TYPE ST_pcmChillerDefaultParameters :
STRUCT
	aSetPointLimitsTemperature : ARRAY[1..2] OF REAL := [10,28];
END_STRUCT
END_TYPE

(* stored: Version 1.1.0.1, ProductVersion 3.1.4024.10
   DUT ST_pcmChillerDefaultParameters: Id {1bf52fc5-d5e5-414f-a4b5-4f031fa292ef} *)
